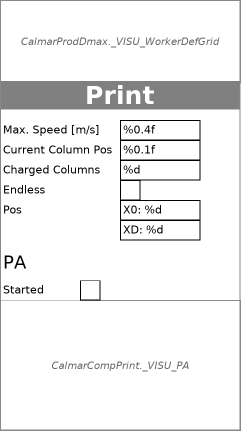
VISUALIZATION _VISU_WorkerPrint_WEU  // 241x431
VAR_IN_OUT
  m_Inst : FB_WorkerDefGrid_Print_WEU;
END_VAR
    Frame (0,0 241x83)
        shows CalmarProdDmax._VISU_WorkerDefGrid(m_Inst := m_Inst)
    Rectangle (0,80 240x30), "Print", colour toggle: m_Inst._pAttachedCt <> 0
    Frame (0,300 241x131)
        shows CalmarCompPrint._VISU_PA(m_Inst := m_Inst.fbPa)
    Rectangle (0,120 120x20), "Max. Speed [m/s]"
    Rectangle (120,120 80x20), "%0.4f", text variable: m_Inst.fMaxSpeed
    Rectangle (0,140 120x20), "Current Column Pos"
    Rectangle (120,140 80x20), "%0.1f", text variable: m_Inst.fCurrentColumnPos
    Rectangle (0,160 120x20), "Charged Columns"
    Rectangle (120,160 80x20), "%d", text variable: m_Inst.nChargedColumns
    Rectangle (0,180 120x20), "Endless"
    RoundedRectangle (120,180 20x20), colour toggle: m_Inst._bEndless
    Rectangle (0,280 80x20), "Started"
    RoundedRectangle (80,280 20x20), colour toggle: m_Inst._bPaStarted
    Rectangle (0,200 120x20), "Pos"
    Rectangle (120,200 80x20), "X0: %d", text variable: m_Inst._nPosX0
    Rectangle (120,220 80x20), "XD: %d", text variable: m_Inst._nPosXDelta
    Rectangle (0,250 240x30), "PA"
END_VISUALIZATION

(* stored: Version 1.1.0.1, ProductVersion 3.1.4024.11
   Visu _VISU_WorkerPrint_WEU: Id {106bf08b-3246-4506-8c48-e81ae7b17b40} *)
